INTERFACE I_AxisJog EXTENDS I_Base

METHOD Jog
VAR_INPUT
	JogForward	 : BOOL;
	JogBackwards : BOOL;
	Position	 : LREAL	 := 0;
END_VAR
END_METHOD

END_INTERFACE

(* stored: Version 1.1.0.1, ProductVersion 3.1.4026.20
   Itf I_AxisJog: Id {df992832-c980-4799-ae8c-2a3f663445af}
   Method Jog: Id {b693a4f3-d11a-4b29-bf9b-3b60c35546a3} *)
